{attribute 'GeneratedUsingTerminal: EL3446-0000-0016'}
{attribute addProperty BoxType "EL3446-0000-0016"}
{attribute addProperty Id "OvercurrentAT %I*BOOL1Inaccurate_CurrentAT %I*BOOL1Current_Guard_WarningAT %I*BOOL1Current_Guard_ErrorAT %I*BOOL1TxPDO_ToggleAT %I*BOOL1CurrentAT %I*REAL4"}
{attribute addProperty CRC "2950815650"}
{attribute addProperty Size "9"}
TYPE I4_Current_AFE1DFA2 EXTENDS InputBase_8311D824 :
STRUCT
	{attribute addProperty Name "Overcurrent"}
	Overcurrent AT %I* : BOOL;
	{attribute addProperty Name "Inaccurate_Current"}
	Inaccurate_Current AT %I* : BOOL;
	{attribute addProperty Name "Current_Guard_Warning"}
	Current_Guard_Warning AT %I* : BOOL;
	{attribute addProperty Name "Current_Guard_Error"}
	Current_Guard_Error AT %I* : BOOL;
	{attribute addProperty Name "TxPDO_Toggle"}
	TxPDO_Toggle AT %I* : BOOL;
	{attribute addProperty Name "Current"}
	Current AT %I* : REAL;
END_STRUCT
END_TYPE

(* stored: Version 1.2.0.0, ProductVersion 3.1.4024.11
   DUT I4_Current_AFE1DFA2: Id {16e7f458-cab7-4839-8159-7dbe4af4a523} *)
